// TIA Portal project "PlcProjekt" (V17)

(* hardware
DEVICE "S7-1200-Station_1"  S7-1200 Station
   slot 0: "Baugruppenträger_0"  S7-1200 Rack  Rack  V1.0
   slot 1: "PLC_1"  CPU 1214C DC/DC/DC  6ES7 214-1AG40-0XB0  V4.2
   slot 3: "AQ 1x12BIT_1"  AQ1 signal board  6ES7 232-4HA30-0XB0  V1.0
*)

// ===== PLC "PLC_1"  CPU 1214C DC/DC/DC =====

VAR_GLOBAL   // PLC tag table "Standard-Variablentabelle"
   "System_Byte" AT %MB100 : Byte;
   "FirstScan" AT %M100.0 : Bool;
   "DiagStatusUpdate" AT %M100.1 : Bool;
   "AlwaysTRUE" AT %M100.2 : Bool;
   "AlwaysFALSE" AT %M100.3 : Bool;
   "Clock_Byte" AT %MB110 : Byte;
   "Clock_10Hz" AT %M110.0 : Bool;
   "Clock_5Hz" AT %M110.1 : Bool;
   "Clock_2.5Hz" AT %M110.2 : Bool;
   "Clock_2Hz" AT %M110.3 : Bool;
   "Clock_1.25Hz" AT %M110.4 : Bool;
   "Clock_1Hz" AT %M110.5 : Bool;
   "Clock_0.625Hz" AT %M110.6 : Bool;
   "Clock_0.5Hz" AT %M110.7 : Bool;
   "ASCII" AT %IB32 : Byte;   // ASCII Code des Zeichens
   "P1R" AT %Q0.0 : Bool;   // Zeiger 1 - Rechts
   "P1L" AT %Q0.1 : Bool;   // Zeiger 1 - Links
   "P2R" AT %Q0.2 : Bool;   // Zeiger 2 - Rechts
   "P2L" AT %Q0.3 : Bool;   // Zeiger 2 - Links
   "P3R" AT %Q0.4 : Bool;   // Zeiger 3 - Rechts
   "P3L" AT %Q0.5 : Bool;   // Zeiger 3 - Links
   "P4R" AT %Q0.6 : Bool;   // Zeiger 4 - Rechts
   "P4L" AT %Q0.7 : Bool;   // Zeiger 4 - Links
   "P5R" AT %Q1.0 : Bool;   // Zeiger 5 - Rechts
   "P5L" AT %Q1.1 : Bool;   // Zeiger 5 - Links
   "ZeigerLowByte" AT %QB0 : Byte;   // Alle Zeiger Low Byte
   "ZeigerHighByte" AT %QB1 : Byte;   // Alle Zieger High Byte
END_VAR

DATA_BLOCK "PcToPlc"   // DB1
{ S7_Optimized_Access := 'FALSE' }
VERSION : 0.1
   VAR
      Plc : Array[0..256] of Byte;
   END_VAR
BEGIN
END_DATA_BLOCK

DATA_BLOCK "PlcToPc"   // DB2
{ S7_Optimized_Access := 'FALSE' }
VERSION : 0.1
   VAR
      Plc : Array[0..256] of Byte;
   END_VAR
BEGIN
END_DATA_BLOCK

DATA_BLOCK "DeleteMe_DB"   // DB3
{ S7_Optimized_Access := 'TRUE' }
VERSION : 0.1
// stored: InstanceOfName DeleteMe
"DeleteMe"
BEGIN
END_DATA_BLOCK

FUNCTION_BLOCK "DeleteMe"   // FB1, SCL
{ S7_Optimized_Access := 'TRUE' }
VERSION : 0.1
   VAR
      Bitmuster : Array[0..256] of Word;
      Init : Bool;
      Zeiger : Int;
      Ergebnis : Word;
   END_VAR
   VAR CONSTANT
      P1R : Word := 2#0000_0000_0001;
      P1L : Word := 2#0000_0000_0010;
      P2R : Word := 2#0000_0000_0100;
      P2L : Word := 2#0000_0000_1000;
      P3R : Word := 2#0000_0001_0000;
      P3L : Word := 2#0000_0010_0000;
      P4R : Word := 2#0000_0100_0000;
      P4L : Word := 2#0000_1000_0000;
      P5R : Word := 2#0001_0000_0000;
      P5L : Word := 2#0010_0000_0000;
   END_VAR
BEGIN
END_FUNCTION_BLOCK

FUNCTION "DatenRangieren" : Void   // FC1, SCL
{ S7_Optimized_Access := 'TRUE' }
VERSION : 0.1
   VAR_TEMP
      TextLaenge : UInt;
   END_VAR
BEGIN
   // Area 16#81 --> Input
   // Area 16#82 --> Output
   // Area 16#84 --> DB

   POKE(area := 16#81,                     // DI (Hardware PLC)
        dbNumber := 0,
        byteOffset := 32,
        value := PEEK(area := 16#84, dbNumber := 1, byteOffset := 32));    // AI des Digital Twin lesen


   // DQ werden immer zum PC übertragen
   POKE(area := 16#84,                         // Datenbausteine
        dbNumber := 2,                         // DB1 -> Pc2Plc
        byteOffset := 0,
        value := PEEK(area := 16#82, dbNumber := 0, byteOffset := 0));

   POKE(area := 16#84,                         // Datenbausteine
        dbNumber := 2,                         // DB1 -> Pc2Plc
        byteOffset := 1,
        value := PEEK(area := 16#82, dbNumber := 0, byteOffset := 1));

   Strg_TO_Chars(Strg := 'Nadeltelegraph V3.0',
                 pChars := 96,
                 Cnt => #TextLaenge,
                 Chars := "PlcToPc".Plc);
END_FUNCTION

ORGANIZATION_BLOCK "Main"   // OB1, LAD, ProgramCycle
TITLE = "Main Program Sweep (Cycle)"
{ S7_Optimized_Access := 'TRUE' }
VERSION : 0.1
   VAR_INPUT
      Initial_Call : Bool;   // Initial call of this OB
      Remanence : Bool;   // =True, if remanent data are available
   END_VAR
BEGIN

REGION Network 1
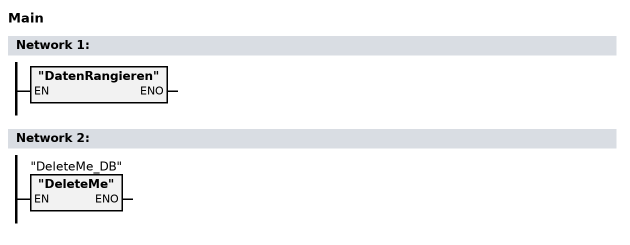
   RUNG wire#powerrail
      "DatenRangieren"()
   END_RUNG
   // the same network as SCL:
   "DatenRangieren"();
END_REGION

REGION Network 2
   RUNG wire#powerrail
      "DeleteMe_DB"()
   END_RUNG
   // the same network as SCL:
   "DeleteMe_DB"();   // "DeleteMe"
END_REGION
END_ORGANIZATION_BLOCK

ORGANIZATION_BLOCK "Startup"   // OB100, SCL, Startup
TITLE = "Complete Restart"
{ S7_Optimized_Access := 'TRUE' }
VERSION : 0.1
   VAR_INPUT
      LostRetentive : Bool;   // True if retentive data are lost
      LostRTC : Bool;   // True if date and time are lost
   END_VAR
BEGIN
   // Area 16#81 --> Input
   // Area 16#82 --> Output
   // Area 16#84 --> DB

   POKE(area := 16#82, dbNumber := 0, byteOffset := 0, value := byte#0);  // Ausgänge löschen
END_ORGANIZATION_BLOCK